// TIA Portal V20 export
// export: Created 2025-12-01T14:57:43.1797279Z, ExportSetting None, DisplayName Totally Integrated Automation Portal, DisplayVersion V20 Update 3, DisplayName TIA Portal Openness, DisplayVersion V20 Update 3, DisplayName TIA Portal Version Control Interface, DisplayVersion V20 Update 3, DisplayName STEP 7 Professional, DisplayVersion V20 Update 3, DisplayName STEP 7 Safety, DisplayVersion V20 Update 2, DisplayName WinCC Basic/Comfort/Advanced, DisplayVersion V20 Update 3, DisplayName WinCC Professional, DisplayVersion V20 Update 3, DisplayName WinCC Unified, DisplayVersion V20 Update 3
DATA_BLOCK "DB1905_RD_IP_GW1"   // DB1905
AUTHOR : SIOS
FAMILY : LPNDR
VERSION : 2.0
// stored: AutoNumber false, InstanceOfName LPNDR_ReadGlobalInfo, InstanceOfType FB
"LPNDR_ReadGlobalInfo"
   // VAR_INPUT
   //    execute : Bool;
   //    hwId : HW_IO;
   // END_VAR
   // VAR_OUTPUT
   //    done { ExternalWritable := 'False'} : Bool;
   //    busy { ExternalWritable := 'False'} : Bool;
   //    error { ExternalWritable := 'False'} : Bool;
   //    status { ExternalWritable := 'False'} : Word;
   //    InterfaceInformation : "LPNDR_typeInterfaceInformation";
   //    PortInformation : Array[1..52] of "LPNDR_typePortInformation";
   //    PortLinkState : Array[1..52] of "LPNDR_typePortLinkState";
   //    PortStatistic : Array[1..52] of "LPNDR_typePortStatistic";
   //    diagnostics { ExternalWritable := 'False'} : "typeDiagnostics";
   // END_VAR
   // VAR
   //    statExecuteOld { ExternalAccessible := 'False'; ExternalVisible := 'False'; ExternalWritable := 'False'} : Bool;
   //    statDone { ExternalAccessible := 'False'; ExternalVisible := 'False'; ExternalWritable := 'False'} : Bool;
   //    statBusy { ExternalAccessible := 'False'; ExternalVisible := 'False'; ExternalWritable := 'False'} : Bool;
   //    statError { ExternalAccessible := 'False'; ExternalVisible := 'False'; ExternalWritable := 'False'} : Bool;
   //    statStatus { ExternalAccessible := 'False'; ExternalVisible := 'False'; ExternalWritable := 'False'} : Word;
   //    statSubfunctionStatus { ExternalAccessible := 'False'; ExternalVisible := 'False'; ExternalWritable := 'False'} : Word;
   //    statFBErrorState { ExternalAccessible := 'False'; ExternalVisible := 'False'; ExternalWritable := 'False'} : DInt;
   //    statFBState { ExternalAccessible := 'False'; ExternalVisible := 'False'; ExternalWritable := 'False'} : DInt;
   //    statEmptyDiagnostics { ExternalAccessible := 'False'; ExternalVisible := 'False'; ExternalWritable := 'False'} : "typeDiagnostics";
   //    InstReadRecord { S7_SetPoint := 'True'} : RDREC;
   //    statReadRecordLength : UInt;
   //    statReadRecordRequest : Bool;
   //    statPDInterfaceMrpDataReal : UInt;
   //    statPDPortMrpDataReal : UInt;
   //    statPDInterfaceDataReal : UInt;
   //    statPDPortDataReal : UInt;
   //    statPDPortStatistic : UInt;
   //    statUnknown : UInt;
   //    statInterfaceInfoReset : "LPNDR_typeInterfaceInformation";
   //    statPortInfoReset { S7_SetPoint := 'True'} : "LPNDR_typePortInformation";
   //    statPortLinkStateReset { S7_SetPoint := 'True'} : "LPNDR_typePortLinkState";
   //    statPortStatisticReset { S7_SetPoint := 'True'} : "LPNDR_typePortStatistic";
   //    statReadRecord { S7_SetPoint := 'True'} : Array[0..4175] of Byte;
   // END_VAR
BEGIN
END_DATA_BLOCK
